# EPICS autosave request: BPMApp/Db/BPMAdcCommon_settings.req
$(P)$(R)ADCTrigDir-Sel
$(P)$(R)ADCTrigTerm-Sel
